{attribute 'GeneratedUsingTerminal: KL6224'}
{attribute addProperty BoxType "KL6224"}
{attribute addProperty Id "Channel_1AT %Q*Channel_08506BCE0"}
{attribute addProperty CRC "3237021629"}
{attribute addProperty Size "0"}
TYPE KL6224_C0F107BD :
STRUCT
	{attribute addProperty Name "Channel_1"}
	Channel_1 : Channel_08506BCE;
END_STRUCT
END_TYPE

(* stored: Version 1.2.0.0, ProductVersion 3.1.4024.9
   DUT KL6224_C0F107BD: Id {4521a0e2-ccdc-4b5f-8565-ba7244070433} *)
